(* CODESYS project ProjectPLC.project

Project tree, tasks and I/O mapping:
  Device : CODESYS Control Win V3 x64, 3S - Smart Software Solutions GmbH, version 3.5.14.20
    application Application
      libraries: Standard, * (System)
      task MainTask (cyclic, interval t#20ms, priority 1) calls PLC_PRG
      program PLC_PRG [LD]
  libraries: VisuSymbols, 3.5.10.0 (System)
  visualisation Visualization
  text list GlobalTextList
*)

// Device/Application/PLC_PRG
PROGRAM PLC_PRG
VAR
	Start: BOOL;
	Stop: BOOL;
	Sensor1: BOOL;
	TON_0: TON;
	Elapsed_Time_Suhu_Detect: TIME;
	TON_1: TON;
	Lampu: BOOL;
	Aktuator: BOOL;
	Elapsed_Time_Aktuator_Mati: TIME;
END_VAR

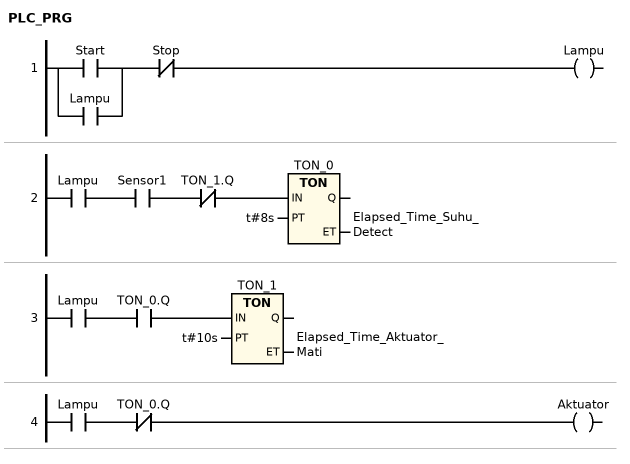
// NETWORK 1
Lampu := (Start OR Lampu) AND NOT Stop;

// NETWORK 2
TON_0(IN := Lampu AND Sensor1 AND NOT TON_1.Q, PT := t#8s, ET => Elapsed_Time_Suhu_Detect); // TON

// NETWORK 3
TON_1(IN := Lampu AND TON_0.Q, PT := t#10s, ET => Elapsed_Time_Aktuator_Mati); // TON

// NETWORK 4
Aktuator := Lampu AND NOT TON_0.Q;

END_PROGRAM

// /Visualization
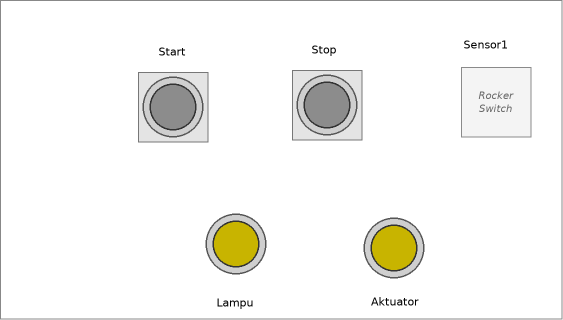
VISUALIZATION Visualization  // 563x320
    PushSwitch (138,72 70x70), variable: PLC_PRG.Start, behaviour: TOGGLE, style: Switch-PushSwitch-Gray
    PushSwitch (292,70 70x70), variable: PLC_PRG.Stop, behaviour: TOGGLE, style: Switch-PushSwitch-Gray
    RockerSwitch (461,67 70x70), variable: PLC_PRG.Sensor1, behaviour: TOGGLE, style: Switch-RockerSwitch-Gray
    Lamp1 (201,209 70x70), variable: PLC_PRG.Lampu, style: Lamp-Lamp1-Yellow
    Lamp1 (359,213 70x70), variable: PLC_PRG.Aktuator, style: Lamp-Lamp1-Yellow
    Label (97,37 150x30), "Start"
    Label (249,35 150x30), "Stop"
    Label (411,30 150x30), "Sensor1"
    Label (160,288 150x30), "Lampu"
    Label (320,287 150x30), "Aktuator"
END_VISUALIZATION
